PROGRAM P06_ProcessControl
VAR CONSTANT
	//Address constants
	HOME			:UINT:=100;
	finish			:UINT:=999;
	done			:UINT:=1000;
	
	//Robot job constants
	//Robot_Pi

END_VAR
VAR_OUTPUT
	q_bAllInHP		:BOOL;
	q_bPause		:BOOL;
END_VAR
VAR
	iStep			:UINT;
END_VAR
VAR // added by the converter: edge detectors and wires of the graphical bodies
    _rt1, _rt2, _rt3, _rt4, _rt5, _rt6, _rt7, _rt8, _rt9, _rt10, _rt11, _rt12 : R_TRIG;
    _w1 : BOOL;
END_VAR

//Select mode
IF Station.stControl.bAuto THEN
	Station.stCommand := Station.stAutoCmd;
ELSIF Station.stControl.bService THEN
	Station.stCommand := Station.stManCmd;
END_IF

//Step-sequence
CASE iStep OF
	0: //Init
	
END_CASE

//Cycle time handler
Station.tonCycleTimer(IN:=(Station.stControl.iStep >= 110 AND Station.stControl.iStep <= 240), PT:=T#10H);

//Shift handler

ACTION GeneralHP:
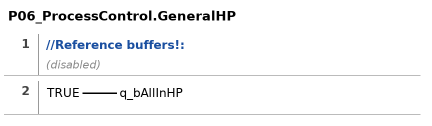
// NETWORK 1 (disabled)
// label: //Reference buffers!

// NETWORK 2
q_bAllInHP := TRUE;
END_ACTION

ACTION PartCounter:
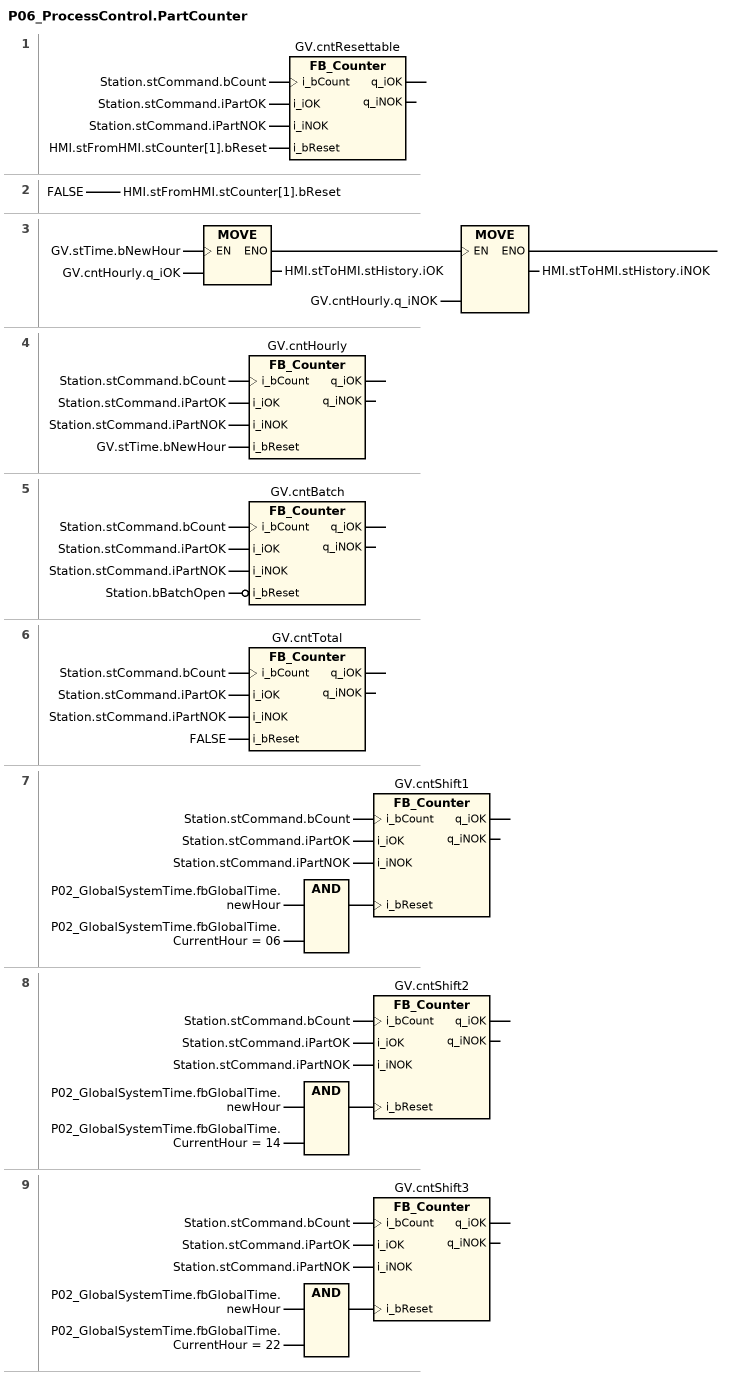
// NETWORK 1
_rt1(CLK := Station.stCommand.bCount);
GV.cntResettable(
    i_bCount := _rt1.Q,
    i_iOK := Station.stCommand.iPartOK,
    i_iNOK := Station.stCommand.iPartNOK,
    i_bReset := HMI.stFromHMI.stCounter[1].bReset); // FB_Counter

// NETWORK 2
HMI.stFromHMI.stCounter[1].bReset := FALSE;

// NETWORK 3
_rt2(CLK := GV.stTime.bNewHour);
_w1 := _rt2.Q;
IF _w1 THEN HMI.stToHMI.stHistory.iOK := GV.cntHourly.q_iOK; END_IF
_rt3(CLK := _w1);
IF _rt3.Q THEN HMI.stToHMI.stHistory.iNOK := GV.cntHourly.q_iNOK; END_IF

// NETWORK 4
_rt4(CLK := Station.stCommand.bCount);
GV.cntHourly(
    i_bCount := _rt4.Q,
    i_iOK := Station.stCommand.iPartOK,
    i_iNOK := Station.stCommand.iPartNOK,
    i_bReset := GV.stTime.bNewHour); // FB_Counter

// NETWORK 5
_rt5(CLK := Station.stCommand.bCount);
GV.cntBatch(
    i_bCount := _rt5.Q,
    i_iOK := Station.stCommand.iPartOK,
    i_iNOK := Station.stCommand.iPartNOK,
    i_bReset := NOT Station.bBatchOpen); // FB_Counter

// NETWORK 6
_rt6(CLK := Station.stCommand.bCount);
GV.cntTotal(
    i_bCount := _rt6.Q,
    i_iOK := Station.stCommand.iPartOK,
    i_iNOK := Station.stCommand.iPartNOK,
    i_bReset := FALSE); // FB_Counter

// NETWORK 7
_rt7(CLK := Station.stCommand.bCount);
_rt8(CLK := P02_GlobalSystemTime.fbGlobalTime.newHour AND (P02_GlobalSystemTime.fbGlobalTime.CurrentHour = 06));
GV.cntShift1(
    i_bCount := _rt7.Q,
    i_iOK := Station.stCommand.iPartOK,
    i_iNOK := Station.stCommand.iPartNOK,
    i_bReset := _rt8.Q); // FB_Counter

// NETWORK 8
_rt9(CLK := Station.stCommand.bCount);
_rt10(CLK := P02_GlobalSystemTime.fbGlobalTime.newHour AND (P02_GlobalSystemTime.fbGlobalTime.CurrentHour = 14));
GV.cntShift2(
    i_bCount := _rt9.Q,
    i_iOK := Station.stCommand.iPartOK,
    i_iNOK := Station.stCommand.iPartNOK,
    i_bReset := _rt10.Q); // FB_Counter

// NETWORK 9
_rt11(CLK := Station.stCommand.bCount);
_rt12(CLK := P02_GlobalSystemTime.fbGlobalTime.newHour AND (P02_GlobalSystemTime.fbGlobalTime.CurrentHour = 22));
GV.cntShift3(
    i_bCount := _rt11.Q,
    i_iOK := Station.stCommand.iPartOK,
    i_iNOK := Station.stCommand.iPartNOK,
    i_bReset := _rt12.Q); // FB_Counter
END_ACTION

ACTION Sequence:

//Control Sequence
CASE Station.stControl.iStep OF
	0: //Initialise : Status - unkonwn
	 	IF Station.stControl.bRunning THEN
		  GeneralHP();
	 	END_IF
		IF q_bAllInHP THEN
			q_bPause := TRUE;
			Station.stControl.iStep := HOME;
		END_IF
		
	
	HOME: //Home : All actuators in HP, wait for START
		Station.stControl.iStep_Prev := 0;
		q_bPause := FALSE;
		GeneralHP();
		IF Station.stControl.bRunning THEN
			Station.stControl.iStep := 110;
		END_IF
		
	110: //Start feeder
		//IF feebdack ok go 200
		
	200: //Buffer Sequence
		//Check input buffer
		IF IN.bSensor_TrayInReady THEN //OK path
			Station.stControl.iStep_Prev := Station.stControl.iStep;
			Station.stControl.iStep := 300;
		ELSE //NOK path
			Station.stControl.iStep_Prev := Station.stControl.iStep;
			Station.stControl.iStep := 210;
			;
		END_IF
	
	210: //Actuate buffer 
		//IF buffer actuation done go 220
	
	220: //Check buffer supply
		//IF buffer position 10 and NOT IN.bSensor_TrayInReady go done
		//IF buffer position <= 10 go 200
		
	300: //Convey carrier
		//IF IN.bSensor_TrayInPick and IN.bSensor_TrayInPlace go 400
		
	400://Robot start
		//In tray position ++
		//Robot job: pick up parts
		//IF Robot feedback OK go 430
		//IF Robot feecback NOK go 420
	
	420://Record missing piece in tray
		//Go to 430
	
	430://Greasing sequence
		//Robot Job := go to greasing
		//IF Robot feedback ok go to 440
	
	440://Grease 
		//IF Greaser feedback ok go 450
	
	450://Turn for greasing
		//Robot Job := turn for greasing
		//IF Robot feedback ok go 460:
	
	460://Grease
		//IF Greaser feedback ok go 500
		
	500://Push BBs to jig
		//IF feedback ok go 600
		//Have a timer for when next push is available	
	
	600://Inspect BB pick position
		//Camera Job := inspect pick BBs
		//IF Job Result OK go 700
		//IF Job Result NOK go 500
	
	700://Attatch BBs
		//Robot Job := attatch BBs
		//IF Robot feedback ok go 800
	
	800://Inspect attatched BBs
		//Camera job := inspect attatched BBs
		//IF Job OK go 900 ELSE go 810
	
	810://Discard bad pats
		//Robot job: discard bad parts
		//IF Robot feedback OK go 900
		
	900://Place done piecese in tray
		//Robot job := place parts
		//IF Robot feedback OK go 910
		
	910://
		
	finish: //Cycle finished: count parts and reset robot
		PartCounter();
		Station.stCommand.bCount := FALSE;
		//IF Robot feedback ok go 120
END_CASE
END_ACTION

END_PROGRAM

(* stored: Version 1.1.0.1
   POU P06_ProcessControl: Id {ef6282b9-d564-4713-9e0c-bcbe889a0ba8}, SpecialFunc None
   Folder Steps: Id {1b752e0e-31c8-46e3-88cc-b55ee095d594}
   Action GeneralHP: Id {9db4dee3-1c67-4104-a4ff-a587859af733}
   Action PartCounter: Id {c33c2f3a-58bc-4b14-a40d-bc4abdfbf757}
   Action Sequence: Id {631d0349-2a91-4c57-901b-cfe65942d6e1} *)
